{attribute 'GeneratedUsingTerminal: EL3008-0000-0017'}
{attribute addProperty BoxType "EL3008-0000-0017"}
{attribute addProperty Id "AI_Standard_Channel_1AT %I*AI_Standard_Channel_4A3944819AI_Standard_Channel_2AT %I*AI_Standard_Channel_4A3944819AI_Standard_Channel_3AT %I*AI_Standard_Channel_4A3944819AI_Standard_Channel_4AT %I*AI_Standard_Channel_4A3944819AI_Standard_Channel_5AT %I*AI_Standard_Channel_4A3944819AI_Standard_Channel_6AT %I*AI_Standard_Channel_4A3944819AI_Standard_Channel_7AT %I*AI_Standard_Channel_4A3944819AI_Standard_Channel_8AT %I*AI_Standard_Channel_4A3944819WcStateAT %I*WcState_9091E0EB2InfoDataAT %I*InfoData_94A18F5E2"}
{attribute addProperty CRC "4233674966"}
{attribute addProperty Size "76"}
TYPE EL3008_FC58C0D6 EXTENDS EtcSlaveTerminalBase_947E5A46 :
STRUCT
	{attribute addProperty Name "AI_Standard_Channel_1"}
	AI_Standard_Channel_1 : AI_Standard_Channel_4A394481;
	{attribute addProperty Name "AI_Standard_Channel_2"}
	AI_Standard_Channel_2 : AI_Standard_Channel_4A394481;
	{attribute addProperty Name "AI_Standard_Channel_3"}
	AI_Standard_Channel_3 : AI_Standard_Channel_4A394481;
	{attribute addProperty Name "AI_Standard_Channel_4"}
	AI_Standard_Channel_4 : AI_Standard_Channel_4A394481;
	{attribute addProperty Name "AI_Standard_Channel_5"}
	AI_Standard_Channel_5 : AI_Standard_Channel_4A394481;
	{attribute addProperty Name "AI_Standard_Channel_6"}
	AI_Standard_Channel_6 : AI_Standard_Channel_4A394481;
	{attribute addProperty Name "AI_Standard_Channel_7"}
	AI_Standard_Channel_7 : AI_Standard_Channel_4A394481;
	{attribute addProperty Name "AI_Standard_Channel_8"}
	AI_Standard_Channel_8 : AI_Standard_Channel_4A394481;
	{attribute addProperty Name "WcState"}
	WcState : WcState_9091E0EB;
	{attribute addProperty Name "InfoData"}
	InfoData : InfoData_94A18F5E;
END_STRUCT
END_TYPE

(* stored: Version 1.2.0.0, ProductVersion 3.1.4024.9
   DUT EL3008_FC58C0D6: Id {a8a03373-7fad-44e1-952f-c451e75c26f5} *)
